// TIA Portal V19 export
FUNCTION_BLOCK "Lubr_Bordat"   // FB121, LAD
// stored: MemoryReserve 100, SetENOAutomatically false
   VAR
      Ton_Stop : TON_TIME;
      Ton_Start : TON_TIME;
      Ctrl { S7_SetPoint := 'True'} : Bool;
      Abilita : Bool;
   END_VAR
BEGIN

REGION Network 1
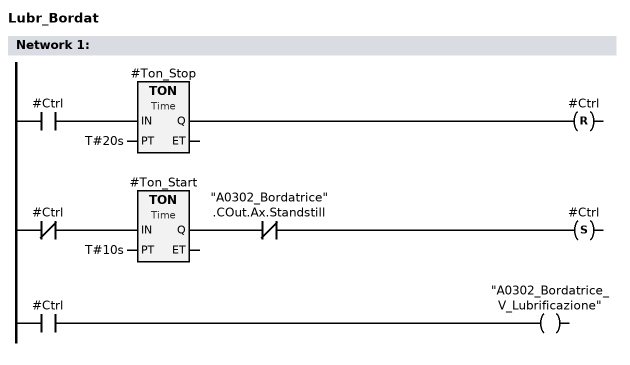
   RUNG wire#powerrail
      Contact( #Ctrl )
      { S7_Templates := "time_type := Time" } #Ton_Stop.TON(pt := T#20s, et =>)
      R_Coil( #Ctrl )
   END_RUNG
   RUNG wire#powerrail
      I_Contact( #Ctrl )
      { S7_Templates := "time_type := Time" } #Ton_Start.TON(pt := T#10s, et =>)
      I_Contact( "A0302_Bordatrice".COut.Ax.Standstill )
      S_Coil( #Ctrl )
   END_RUNG
   RUNG wire#powerrail
      Contact( #Ctrl )
      Coil( "A0302_Bordatrice_V_Lubrificazione" )
   END_RUNG
   // the same network as SCL:
   #Ton_Stop(IN := #Ctrl, PT := T#20s);   // TON
   IF #Ton_Stop.Q THEN #Ctrl := FALSE; END_IF;
   #Ton_Start(IN := NOT #Ctrl, PT := T#10s);   // TON
   IF #Ton_Start.Q AND NOT "A0302_Bordatrice".COut.Ax.Standstill THEN #Ctrl := TRUE; END_IF;
   "A0302_Bordatrice_V_Lubrificazione" := #Ctrl;
END_REGION
END_FUNCTION_BLOCK
